# EPICS substitutions: iocBoot/ioc-xrt-xcsimb1/ioc-xrt-xcsimb1.substitutions
# IOC archive file
## Replace XRT:R04:IOC:35 with the PV prefix used for
## iocAdmin PV's on this IOC

# Generate IOC archive request
file archive_ipimbIoc.archive
{
	{ IOC = "XRT:R04:IOC:35" }
}
